Staubli VAL3: duplicate.pgx

public program duplicate(string x_sCopy, string x_sPaste, num& x_nResult[])
  local num i
  local num l_nSize
  local string l_sItem
  local bool l_bFound
  local num l_nResult
  local string l_sString
  local num l_nX
  local num l_nY
begin
  // duplicate

  // look if the items exist
  if insert(pt:tTraj[x_sPaste])
    // link the point
    call pt:copy_it(x_sCopy,x_sPaste)
    call pt:link_all(x_sPaste)
    // save it
    bToSave=true
  endIf
end
